INTERFACE I_ChunkedRequestsHeaderAccessor

METHOD PUBLIC TryGetChunkSequenceFromRequest : BOOL
VAR_INPUT
	Request : I_Request;
	Destination : REFERENCE TO DINT;
END_VAR
END_METHOD

METHOD PUBLIC TryGetChunkTotalFromRequest : BOOL
VAR_INPUT
	Request : I_Request;
	Destination : REFERENCE TO DINT;
END_VAR
END_METHOD

METHOD PUBLIC TryGetHasMoreChunksFromRequest : BOOL
VAR_INPUT
	Request : I_Request;
	Destination : REFERENCE TO BOOL;
END_VAR
END_METHOD

METHOD PUBLIC TryGetRequestIdFromRequest : BOOL
VAR_INPUT
	Request : I_Request;
	Destination : REFERENCE TO T_MAXSTRING;
END_VAR
END_METHOD

METHOD PUBLIC TryGetSessionIdFromRequest : BOOL
VAR_INPUT
	Request : I_Request;
	Destination : REFERENCE TO T_MAXSTRING;
END_VAR
END_METHOD

END_INTERFACE

(* stored: Version 1.1.0.1, ProductVersion 3.1.4024.12
   Itf I_ChunkedRequestsHeaderAccessor: Id {e908ebff-30b2-0e47-1ddd-740471b4efb3}
   Method TryGetChunkSequenceFromRequest: Id {edb39f6f-fadf-0ff8-0d84-5852df9fe9ea}
   Method TryGetChunkTotalFromRequest: Id {84948862-eb2e-0c4e-2599-3af4eba93d74}
   Method TryGetHasMoreChunksFromRequest: Id {e4fa4ddf-77bf-0116-398e-94c3b772b9cb}
   Method TryGetRequestIdFromRequest: Id {a82fb7c8-9f8a-0813-39f5-0bc72b582830}
   Method TryGetSessionIdFromRequest: Id {68258ed8-7502-0250-33ff-2a144e7ddc94} *)
